// TIA Portal V19 export
TYPE "C501_STU_IF_KLG_TYPIC"
   STRUCT
      CMD { ExternalAccessible := 'False'; ExternalVisible := 'False'; ExternalWritable := 'False'} : Bool;   // Aansturing klep (TRUE = Open / FALSE = Toe)
      CMD_RES { ExternalAccessible := 'False'; ExternalVisible := 'False'; ExternalWritable := 'False'} : Bool;   // Reset van de latched storingen
   END_STRUCT;
END_TYPE
